{attribute 'qualified_only'}
{attribute 'strict'}
(*Вид аварийной блокировки*)
TYPE AlarmType :
(
	Alarm_LocalQuit 	:= 0,
	Alarm_ScadaQuit 	:= 1,
	Alarm_NoQuit 		:= 2,
	Warning_RecordOnly	:= 3,
	Warning_Type2		:= 4
);
END_TYPE

(* stored: Version 1.1.0.1, ProductVersion 3.1.4022.10
   DUT AlarmType: Id {9b12f8e9-6cb4-4048-b044-3ce567f881a6} *)
